FUNCTION_BLOCK ROBOT_LD90 EXTENDS FB_2_ROB_AMR

END_FUNCTION_BLOCK

(* stored: Version 1.1.0.1, ProductVersion 3.1.4026.18
   POU ROBOT_LD90: Id {fac74160-c2b3-4f77-bd69-eddf1970c653}, SpecialFunc None *)
